/// configuration data that is used during boot to configure the Units equipment
TYPE XyTableDataConfig :
STRUCT
  Simulated : BOOL;
END_STRUCT
END_TYPE

(* stored: Version 1.1.0.1
   DUT XyTableDataConfig: Id {2d1a4b21-7f2e-405f-aabf-66e05fcec3e6} *)
